FUNCTION_BLOCK AX_AND_6 (* FB to calculate boolean AND (generic FB) Adapter-Ausgang wird nur bei Wertänderung aktualisiert (Event nur bei tatsächlicher Änderung). *)
  (* Standard: 61499-2; Description: Copyright (c) 2024 HR Agrartechnik GmbH This program and the accompanying materials are made available under the terms of the Eclipse Public License 2.0 which is available at https://www.eclipse.org/legal/epl-2.0/ SPDX-License-Identifier: EPL-2.0 *)
  (* Version 1.0, 2026-09-17, Franz Höpfinger, HR Agrartechnik GmbH, Neu (Franz: 'AX_AND_6 einfach anlegen, das ist ein GEN-FB, das geht so') - fuer die Not-Halt-Sammelueberwachung (STG1 I1-I6) auf der Launch-Page, analog AX_AND_2/AX_AND_3/AX_AND_4. *)
  PACKAGE adapter::booleanOperators;
  IMPORT eclipse4diac::core::GenericClassName;
  {SET_ATTRIBUTE(eclipse4diac::core::GenericClassName, 'GEN_AX_AND')}
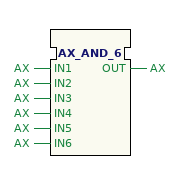
  SOCKETS
    IN1 : adapter::types::unidirectional::AX; (* AND input 1 *)
    IN2 : adapter::types::unidirectional::AX; (* AND input 2 *)
    IN3 : adapter::types::unidirectional::AX; (* AND input 3 *)
    IN4 : adapter::types::unidirectional::AX; (* AND input 4 *)
    IN5 : adapter::types::unidirectional::AX; (* AND input 5 *)
    IN6 : adapter::types::unidirectional::AX; (* AND input 6 *)
  END_SOCKETS
  PLUGS
    OUT : adapter::types::unidirectional::AX; (* AND result *)
  END_PLUGS
END_FUNCTION_BLOCK
